INTERFACE ITF_Control2 EXTENDS ITF_BaseControlElement

END_INTERFACE

(* stored: Version 1.1.0.1
   Itf ITF_Control2: Id {c9fc5188-8463-043c-1143-0f2b63ddef3a} *)
